PROGRAM MAIN
VAR
END_VAR

Alias();
//Heartbeat();
Permissives();
Trips();
Alarms();
Sequence();
Communication();
Analogconversion();
HMI();
ChargeTime();

END_PROGRAM

(* stored: Version 1.1.0.1, ProductVersion 3.1.4024.11
   POU MAIN: Id {d2269fb9-f8e5-4fd2-b745-5dc1f350dc3d}, SpecialFunc None *)
